INTERFACE I_ControlBox

METHOD Joy_Normalized : REAL
VAR_INPUT
	JoyX_raw : LREAL;
	JoyY_raw : LREAL;
END_VAR
VAR_OUTPUT
	JoyX_normalized : LREAL;
	JoyY_normalized : LREAL;
END_VAR
END_METHOD

METHOD Mode
VAR_OUTPUT
	eMode : E_Control_Mode;
END_VAR
END_METHOD

METHOD Status : E_Status
VAR_INPUT
	eMode : E_Control_Mode;
	bStartButton : BOOL;
	bStopButton: BOOL;
END_VAR
VAR_OUTPUT
	sControlMode : STRING;
END_VAR
END_METHOD

END_INTERFACE

(* stored: Version 1.1.0.1, ProductVersion 3.1.4024.12
   Itf I_ControlBox: Id {9f885559-3305-4675-809f-2cf4e90fe19b}
   Method Joy_Normalized: Id {5d4130d3-6c3a-4ac5-9965-d1fc49c0529c}
   Method Mode: Id {c5c82611-b5c0-4eb8-9171-b21927bf4a1d}
   Method Status: Id {5107072e-e81b-4166-af85-2c0de74e031a} *)
